// TIA Portal V19 export
DATA_BLOCK "DB_Sperrbereiche"   // DB68
{ S7_Optimized_Access := 'FALSE' }
// stored: AutoNumber false
   VAR RETAIN
      Anzahl : Int := 4;   // * Anzahl der definierten Sperrbereiche
      resD : DInt := 0;
      resw : Int := 0;
      DG1_aktiv : Bool := FALSE;
      DG1_Quit : Bool := FALSE;
      DG1_FP_Taste : Bool := FALSE;
      DG1_Req : Bool := FALSE;
      DG2_aktiv : Bool := FALSE;
      DG2_Quit : Bool := FALSE;
      DG2_FP_Taste : Bool := FALSE;
      DG2_Req : Bool := FALSE;
      Sperre_links : Bool := FALSE;
      Sperre_rechts : Bool := FALSE;
      res3 : Bool := FALSE;
      res4 : Bool := FALSE;
      res5 : Bool := FALSE;
      res6 : Bool := FALSE;
      res7 : Bool := FALSE;
      res8 : Bool := FALSE;
      Bereich : Array[1..5] of Struct   // * Feldlänge anpassen
         aktiv : Bool;   // Bereich ist gesperrt
         min_Inc : DInt;   // untere Grenze Sperrbereich
         max_Inc : DInt;   // obere Grenze Sperrbereich
      END_STRUCT;
   END_VAR
BEGIN
   Bereich[1..5].aktiv := FALSE;
   Bereich[1].min_Inc := 1242;
   Bereich[2].min_Inc := 4938;
   Bereich[3].min_Inc := 1242;
   Bereich[4].min_Inc := 4130;
   Bereich[5].min_Inc := 0;
   Bereich[1].max_Inc := 3372;
   Bereich[2].max_Inc := 7901;
   Bereich[3].max_Inc := 4100;
   Bereich[4].max_Inc := 8654;
   Bereich[5].max_Inc := 0;
END_DATA_BLOCK
